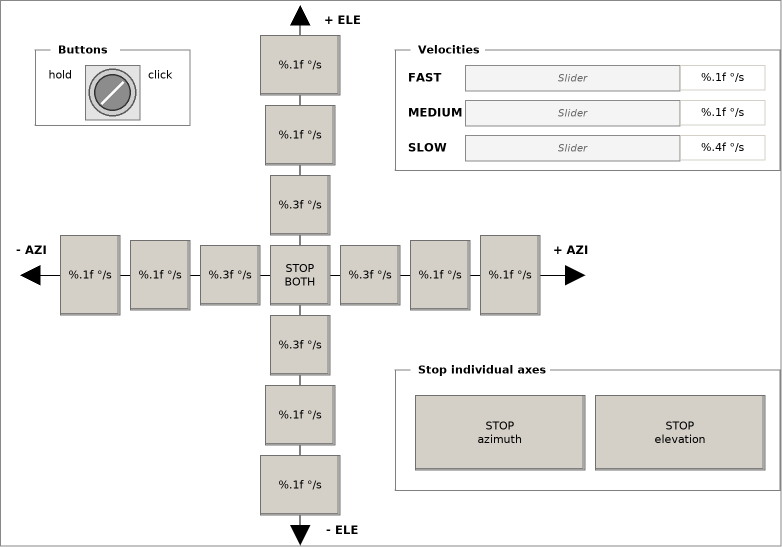
VISUALIZATION VISU_AxesManual_Joystick_AziEle  // 782x547
VAR_IN_OUT
	ref : Axes;
    widget : AxesManualJoystickAziEleWidget;
END_VAR
    Polyline (410,50) (395,50) (395,170) (780,170) (780,50) (485,50)
    Line (40,275) (575,275)
    Line (300,525) (300,25)
    Slider (465,65 215x26), variable: widget.joystick_velocity_fast, input disabled if: widget.joystick_disabled, scale 0..3
    Button (260,35 80x60), "%.1f °/s", text variable: widget.joystick_velocity_fast, input disabled if: widget.jog_ele_disabled
        tap widget.jog_ele_forward_fast
    Button (265,105 70x60), "%.1f °/s", text variable: widget.joystick_velocity_medium, input disabled if: widget.jog_ele_disabled
        tap widget.jog_ele_forward_medium
    Button (270,175 60x60), "%.3f °/s", text variable: widget.joystick_velocity_slow, input disabled if: widget.jog_ele_disabled
        tap widget.jog_ele_forward_slow
    Button (270,245 60x60), "STOP BOTH", input disabled if: ref.processes.stop.statuses.enabledStatus.disabled
        OnMouseClick: execute { ref.processes.stop.request(); }
    Button (260,455 80x60), "%.1f °/s", text variable: widget.joystick_velocity_fast, input disabled if: widget.jog_ele_disabled
        tap widget.jog_ele_backwards_fast
    Button (265,385 70x60), "%.1f °/s", text variable: widget.joystick_velocity_medium, input disabled if: widget.jog_ele_disabled
        tap widget.jog_ele_backwards_medium
    Button (270,315 60x60), "%.3f °/s", text variable: widget.joystick_velocity_slow, input disabled if: widget.jog_ele_disabled
        tap widget.jog_ele_backwards_slow
    Button (200,245 60x60), "%.3f °/s", text variable: widget.joystick_velocity_slow, input disabled if: widget.jog_azi_disabled
        tap widget.jog_azi_backwards_slow
    Button (130,240 60x70), "%.1f °/s", text variable: widget.joystick_velocity_medium, input disabled if: widget.jog_azi_disabled
        tap widget.jog_azi_backwards_medium
    Button (60,235 60x80), "%.1f °/s", text variable: widget.joystick_velocity_fast, input disabled if: widget.jog_azi_disabled
        tap widget.jog_azi_backwards_fast
    Button (480,235 60x80), "%.1f °/s", text variable: widget.joystick_velocity_fast, input disabled if: widget.jog_azi_disabled
        tap widget.jog_azi_forward_fast
    Button (410,240 60x70), "%.1f °/s", text variable: widget.joystick_velocity_medium, input disabled if: widget.jog_azi_disabled
        tap widget.jog_azi_forward_medium
    Button (340,245 60x60), "%.3f °/s", text variable: widget.joystick_velocity_slow, input disabled if: widget.jog_azi_disabled
        tap widget.jog_azi_forward_slow
    Textfield (680,65 85x25), "%.1f °/s", text variable: widget.joystick_velocity_fast, input disabled if: widget.joystick_disabled
        OnMouseClick: write the text variable via VisuDialogs.Numpad, min 0, max 3
    Polygon (290,25) (300,5) (310,25)
    Polygon (290,525) (300,545) (310,525)
    Polygon (565,285) (565,265) (585,275)
    Polygon (40,285) (40,265) (20,275)
    Label (405,65 70x25), "FAST"
    Slider (465,100 215x26), variable: widget.joystick_velocity_medium, input disabled if: widget.joystick_disabled, scale 0..3
    Label (405,100 70x25), "MEDIUM"
    Slider (465,135 215x26), variable: widget.joystick_velocity_slow, input disabled if: widget.joystick_disabled, scale 0..3
    Label (405,135 70x25), "SLOW"
    Label (415,40 70x20), "Velocities"
    Textfield (680,100 85x25), "%.1f °/s", text variable: widget.joystick_velocity_medium, input disabled if: widget.joystick_disabled
        OnMouseClick: write the text variable via VisuDialogs.Numpad, min 0, max 3
    Textfield (680,135 85x25), "%.4f °/s", text variable: widget.joystick_velocity_slow, input disabled if: widget.joystick_disabled
        OnMouseClick: write the text variable via VisuDialogs.Numpad, min 0, max 3
    Label (315,5 55x30), "+ ELE"
    Label (315,515 55x30), "- ELE"
    Label (550,235 45x30), "+ AZI"
    Label (10,235 40x30), "- AZI"
    Label (415,360 135x20), "Stop individual axes"
    Polyline (410,370) (395,370) (395,490) (780,490) (780,370) (550,370)
    Button (415,395 170x75), "STOP azimuth", input disabled if: ref.parts.azi.processes.stop.statuses.enabledStatus.disabled
        OnMouseClick: execute { ref.parts.azi.processes.stop.request(); }
    Button (595,395 170x75), "STOP elevation", input disabled if: ref.parts.ele.processes.stop.statuses.enabledStatus.disabled
        OnMouseClick: execute { ref.parts.ele.processes.stop.request(); }
    Polyline (50,50) (35,50) (35,125) (190,125) (190,50) (120,50)
    RotarySwitch (85,65 55x55), variable: widget.joystick_hold, input disabled if: widget.joystick_disabled, behaviour: TOGGLE, style: Switch-RotarySwitch-Gray
    Label (145,65 50x20), "click"
    Label (35,65 40x20), "hold"
    Label (55,40 65x20), "Buttons"
END_VISUALIZATION

(* stored: Version 1.1.0.1, ProductVersion 3.1.4019.2
   Visu VISU_AxesManual_Joystick_AziEle: Id {c34a81a6-0f65-427e-a973-4b1c9b549c96} *)
